VISUALIZATION AstModel  // 2x2
END_VISUALIZATION

(* stored: Version 1.1.0.1
   Visu AstModel: Id {9f626ebe-0fb9-4a76-9c05-ae1c7221a00f} *)
